FUNCTION_BLOCK FB_Cylinder
VAR_INPUT
	Position_Extend: BOOL;
END_VAR
VAR_OUTPUT
	Status_Extended:BOOL;
END_VAR
VAR
	CylinderOutput AT %Q*:BOOL;
END_VAR

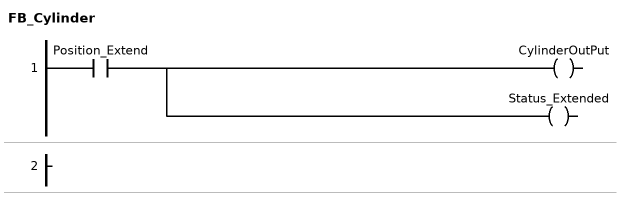
// NETWORK 1
CylinderOutPut := Position_Extend;
Status_Extended := Position_Extend;

// NETWORK 2

END_FUNCTION_BLOCK

(* stored: Version 1.1.0.1, ProductVersion 3.1.4024.4
   POU FB_Cylinder: Id {1c656a5d-6af9-416a-ab6b-7a7a3efe732f}, SpecialFunc None *)
